///#########################################################
///Function block to run a virtual drive with Nc
///	Library:		
///	Tc2_MC2.lib
///
///	Global Variables:
///	
///	Data types:
///	
///	External functions:
///
///###########################################################
FUNCTION_BLOCK FB_Axis
VAR
	sVersion: STRING:='1.0.3';	
	
END_VAR
VAR_INPUT
	bEnable: BOOL;
	bReset: BOOL;
	bExecute: BOOL;
	bStop: BOOL;
	eCommand: MotionFunctions; 
END_VAR
VAR_OUTPUT
	bEnabled: BOOL;
	bBusy: BOOL;
	bDone: BOOL;
	bError: BOOL;
END_VAR

VAR_IN_OUT
	stAxisStruct: ST_AxisStruct;
END_VAR
VAR	
	fbReset: MC_Reset;
	fbPower: MC_Power;
	fbStop: MC_Stop;
	fbHalt: MC_Halt;
	fbJog: MC_Jog;
	fbMoveAbsolute: MC_MoveAbsolute;
	fbMoveVelocity: MC_MoveVelocity;
	fbMoveRelative: MC_MoveRelative;
	fbMoveModulo: MC_MoveModulo;	
	fbGearInDyn: MC_GearInDyn;
	fbGearOut: MC_GearOut;
	fbHome: FB_Homing;
	fbExecuteRiseEdge: R_TRIG;
END_VAR

//Connection of variables to tha Axis Structure//
bExecute:= stAxisStruct.bExecute;
eCommand:=stAxisStruct.eCommand;

////Call of all MC Instances//////

fbPower(Axis:=stAxisStruct.Axis);
fbPower.Enable:= FALSE;
fbReset(Axis:=stAxisStruct.Axis);
fbReset.Execute:= FALSE;
fbStop(Axis:=stAxisStruct.Axis);
fbStop.Execute:=FALSE;
fbHalt(Axis:=stAxisStruct.Axis);
fbHalt.Execute:=FALSE;
fbJog(Axis:=stAxisStruct.Axis);
fbHome(Axis:=stAxisStruct.Axis);
fbHome.bExecute:=FALSE;
fbMoveAbsolute(Axis:=stAxisStruct.Axis);
fbMoveAbsolute.Execute:=FALSE;
fbMoveRelative(Axis:=stAxisStruct.Axis);
fbMoveRelative.Execute:=FALSE;
fbMoveVelocity(Axis:=stAxisStruct.Axis);
fbMoveVelocity.Execute:=FALSE;
fbMoveModulo(Axis:=stAxisStruct.Axis);
fbMoveModulo.Execute:=FALSE;
//fbGearInDyn(Master:=, Slave:=);
fbGearInDyn.Enable:=FALSE;
//fbGearOut(Slave:=);
fbGearOut.Execute:=FALSE;


(*Power*)
	fbPower.Enable:=bEnable;
	fbPower.Enable_Positive:=bEnable AND stAxisStruct.bLimitFwd;	
	fbPower.Enable_Negative:=bEnable AND stAxisStruct.bLimitBwd;
	fbPower.Override:= stAxisStruct.fOverride;
	bEnabled:=fbPower.Status;

(*Stop*)	
	fbStop.Execute:= bStop;
	fbStop.Deceleration:= stAxisStruct.fDeceleration;
				
(*Reset*)
	fbReset.Execute:=bReset AND stAxisStruct.Axis.Status.Error;


CASE eCommand OF
	MotionFunctions.MoveAbsolute:
		fbMoveAbsolute.Execute:=bExecute;
		fbMoveAbsolute.Position:=stAxisStruct.fPosition;
		fbMoveAbsolute.Velocity:=ABS(stAxisStruct.fVelocity);
		fbMoveAbsolute.Acceleration:=stAxisStruct.fAcceleration;
		fbMoveAbsolute.Deceleration:=stAxisStruct.fDeceleration;
				
	MotionFunctions.MoveRelative:
		fbMoveRelative.Execute:=bExecute;
		fbMoveRelative.Distance:=stAxisStruct.fPosition;
		fbMoveRelative.Velocity:=ABS(stAxisStruct.fVelocity);
		fbMoveRelative.Acceleration:=stAxisStruct.fAcceleration;
		fbMoveRelative.Deceleration:=stAxisStruct.fDeceleration;
				
	MotionFunctions.Jog:
		fbJog.JogForward:=stAxisStruct.bJogFwd AND NOT bExecute;
		fbJog.JogBackwards:=stAxisStruct.bJogBwd AND NOT bExecute;
		fbJog.Mode:=0;
		fbJog.Velocity:=stAxisStruct.fVelocity;
		fbJog.Acceleration:=stAxisStruct.fAcceleration;
		fbJog.Deceleration:=stAxisStruct.fDeceleration;
				
	MotionFunctions.MoveVelocity:
		fbMoveVelocity.Execute:=bExecute;
		fbMoveVelocity.Velocity:=ABS(stAxisStruct.fVelocity);
		fbMoveVelocity.Acceleration:=stAxisStruct.fAcceleration;
		fbMoveVelocity.Deceleration:=stAxisStruct.fDeceleration;
		fbMoveVelocity.Direction:=SEL(stAxisStruct.fVelocity<0, MC_Positive_Direction, MC_Negative_Direction);

	MotionFunctions.Movemodulo:
		fbMoveModulo.Execute:=bExecute;
		fbMoveModulo.Position:=stAxisStruct.fPosition;
		fbMoveModulo.Velocity:=ABS(stAxisStruct.fVelocity);
		fbMoveModulo.Acceleration:=stAxisStruct.fAcceleration; 
		fbMoveModulo.Deceleration:=stAxisStruct.fDeceleration;

				
	MotionFunctions.SingleGearIn:
	
	MotionFunctions.SingleGearOut:
	
	MotionFunctions.MultiGear:
			
	MotionFunctions.Home:
		fbHome.bExecute:= bExecute;
		fbHome.bReset:= bReset;
		fbHome.nHomeProc:= stAxisStruct.nHomeSeq;
		fbHome.bLimitBwd:= stAxisStruct.bLimitBwd; 
		fbHome.bLimitFwd:= stAxisStruct.bLimitFwd; 
		fbHome.bEncLatch:= stAxisStruct.bEncLatch;
		fbHome.bHomeSensor:= stAxisStruct.bHomeSensor;
		fbHome.fHomePosition:= 0; 
		stAxisStruct.bHomed:=fbHome.bHomed;
				
END_CASE			


(*Busy*)
bBusy:=stAxisStruct.Axis.Status.HasJob;

(*Error from functions and Nc*)
IF fbPower.Error AND fbPower.Active THEN
	bError:=fbPower.Enable;
	stAxisStruct.nErrorId:=fbPower.ErrorID;
ELSIF fbHalt.Error AND fbHalt.Active THEN
	bError:=fbHalt.Execute;
	stAxisStruct.nErrorId:=fbHalt.ErrorID;
ELSIF fbJog.Error THEN
	bError:=fbJog.JogForward OR fbJog.JogBackwards;
	stAxisStruct.nErrorId:=fbJog.ErrorID;
ELSIF fbMoveVelocity.Error THEN
	bError:=fbMoveVelocity.Execute;
	stAxisStruct.nErrorId:=fbMoveVelocity.ErrorID;
ELSIF fbMoveRelative.Error THEN
	bError:=fbMoveRelative.Execute;
	stAxisStruct.nErrorId:=fbMoveRelative.ErrorID;
ELSIF fbMoveAbsolute.Error THEN
	bError:=fbMoveAbsolute.Execute;
	stAxisStruct.nErrorId:=fbMoveAbsolute.ErrorID;
ELSIF fbMoveModulo.Error THEN
	bError:=fbMoveModulo.Execute;
	stAxisStruct.nErrorId:=fbMoveModulo.ErrorID;
ELSIF fbHome.bError THEN
	bError:=fbHome.bError;
	stAxisStruct.nErrorId:=fbHome.nErrorID;
ELSIF fbGearInDyn.Error THEN
	bError:=fbGearInDyn.Enable;
	stAxisStruct.nErrorId:=fbGearInDyn.ErrorID;
ELSIF fbGearOut.Error and stAxisStruct.Axis.Status.Coupled THEN
	bError:=fbGearOut.Execute;
	stAxisStruct.nErrorId:=fbGearOut.ErrorID;
ELSIF stAxisStruct.Axis.Status.Error  THEN
	bError:=TRUE;
	stAxisStruct.nErrorId:=stAxisStruct.Axis.Status.ErrorID;
ELSE
	bError:=FALSE;
	stAxisStruct.nErrorId:=0;
END_IF;

(*Actual Velocity*)
stAxisStruct.fActVelocity:=stAxisStruct.Axis.NcToPlc.ActVelo;

(*Actual Position*)
IF stAxisStruct.Axis.Status.OpMode.Modulo THEN
	stAxisStruct.fActPosition:=stAxisStruct.Axis.NcToPlc.ModuloActPos;
ELSE
	stAxisStruct.fActPosition:=stAxisStruct.Axis.NcToPlc.ActPos;
END_IF

END_FUNCTION_BLOCK

(* stored: Version 1.1.0.1, ProductVersion 3.1.4022.10
   POU FB_Axis: Id {45901cd0-c6d2-4114-b7cf-de832171219f}, SpecialFunc None *)
